TYPE ST_BhElFlow :
STRUCT
	eFlowUnit	:	E_BHElFlowUnit;
	i_udiUnit	:	UDINT;
	i_rFlow	:	REAL;
END_STRUCT
END_TYPE

(* stored: Version 1.1.0.1, ProductVersion 3.1.4020.12
   DUT ST_BhElFlow: Id {aa56882c-6739-4583-9306-a6edfd4b5ed1} *)
